{attribute addProperty BoxType "EL5072-0000-0016"}
{attribute addProperty Id "Set_positionAT %Q*BOOL811Set_position_on_digital_inputAT %Q*BOOL812Enable_latch_on_digital_inputAT %Q*BOOL813Set_position_valueAT %Q*DINT32417"}
{attribute addProperty CRC "3451475005"}
{attribute addProperty SizeInBites "56"}
{attribute addProperty SizeInBytes "7"}
TYPE IND_Outputs_Channel_CDB9543D :
STRUCT
	{attribute addProperty Name "Set_position"}
	Set_position AT %Q* : BOOL;
	{attribute addProperty Name "Set_position_on_digital_input"}
	Set_position_on_digital_input AT %Q* : BOOL;
	{attribute addProperty Name "Enable_latch_on_digital_input"}
	Enable_latch_on_digital_input AT %Q* : BOOL;
	{attribute addProperty Name "Set_position_value"}
	Set_position_value AT %Q* : DINT;
END_STRUCT
END_TYPE

(* stored: Version 1.2.0.0, ProductVersion 3.1.4024.9
   DUT IND_Outputs_Channel_CDB9543D: Id {eadd1113-ce33-45d3-b900-b90fbd7f47a8} *)
